Yaskawa INFORM job: big_bent_cylinder_program.JBI

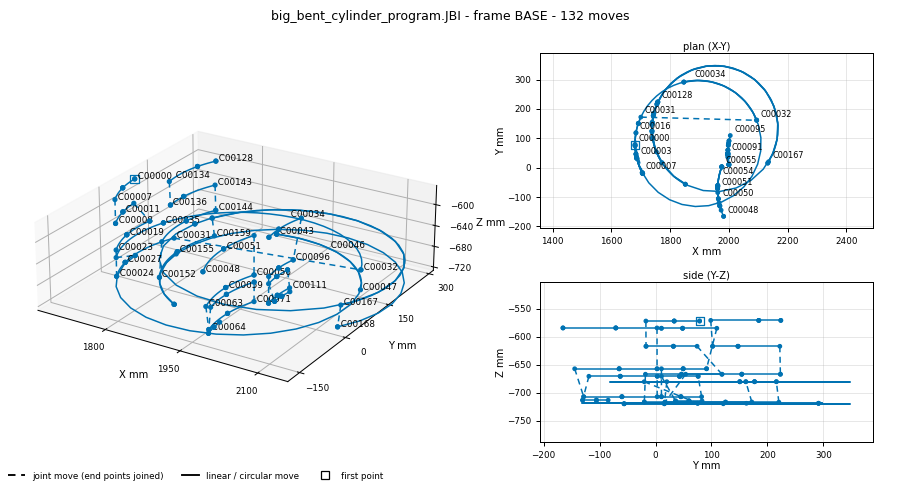
[picture p0: tool path of big_bent_cylinder_program.JBI in frame BASE, 132 of 185 moves have a stored position in this frame; points joined in program order, loops and branches not executed]
/JOB
//NAME big_bent_cylinder_program
//POS
///NPOS 176,0,176,0,0,0
///TOOL 0
///POSTYPE BASE
///RECTAN
///RCONF 0,0,0,0,0,0,0,0,0,0,0,0,0,0,0,0,0,0,0,0,0,0,0,0
C00000=1680.662060,78.729011,-571.725500,-175.000000,-89.999999,5.000000
C00001=1680.662060,78.729011,-571.725500,-175.000000,-89.999999,5.000000
C00002=1681.281377,65.697405,-571.725500,-175.000000,-89.999999,5.000000
C00003=1686.307736,33.361169,-571.725500,-166.791969,-90.000000,5.000000
C00004=1686.307736,33.361169,-571.725500,-166.791969,-90.000000,5.000000
C00005=1686.307736,33.361169,-571.725500,-166.791969,-90.000000,5.000000
C00006=1696.081532,2.440055,-571.725500,-158.125782,-90.000000,5.000000
C00007=1705.179944,-17.274311,-571.725500,-152.326458,-90.000000,5.000000
C00008=1705.056434,-17.038439,-616.865500,-152.397542,-90.000000,5.000000
C00009=1705.056434,-17.038439,-616.865500,-152.397542,-90.000000,5.000000
C00010=1691.809992,14.034424,-616.865500,-161.425103,-90.000000,5.000000
C00011=1686.649002,31.929188,-616.865500,-166.398950,-89.999999,5.000000
C00012=1686.649002,31.929188,-616.865500,-166.398950,-89.999999,5.000000
C00013=1686.649002,31.929188,-616.865500,-166.398950,-89.999999,5.000000
C00014=1685.912600,35.076369,-616.865500,-167.261890,-89.999999,5.000000
C00015=1680.785043,74.259067,-616.865500,-175.000000,-89.999999,5.000000
C00016=1683.724650,118.705496,-666.897500,170.259212,-90.000000,5.000000
C00017=1683.724650,118.705496,-666.897500,170.259212,-90.000000,5.000000
C00018=1682.076679,57.525758,-666.897500,-173.345168,-90.000000,5.000000
C00019=1683.676867,46.365991,-666.897500,-170.334905,-89.999999,5.000000
C00020=1683.676867,46.365991,-666.897500,-170.334905,-89.999999,5.000000
C00021=1683.676867,46.365991,-666.897500,-170.334905,-89.999999,5.000000
C00022=1694.919230,5.398308,-666.897500,-158.974360,-90.000000,5.000000
C00023=1705.611428,-18.092796,-666.897500,-152.079433,-90.000000,5.000000
C00024=1706.664513,-20.055320,-716.487000,-151.484806,-89.999999,5.000000
C00025=1706.664513,-20.055320,-716.487000,-151.484806,-89.999999,5.000000
C00026=1685.911416,35.081606,-716.487000,-167.263323,-89.999999,5.000000
C00027=1685.559141,36.668028,-716.487000,-167.697185,-90.000000,5.000000
C00028=1685.559141,36.668028,-716.487000,-167.697185,-90.000000,5.000000
C00029=1685.559141,36.668028,-716.487000,-167.697185,-90.000000,5.000000
C00030=1681.109891,96.728954,-716.487000,175.000000,-90.000000,5.000000
C00031=1700.273814,172.091124,-716.487000,155.294663,-89.999999,5.000000
C00032=2094.761755,161.426578,-680.269460,175.000000,-60.000000,-158.391764
C00033=2094.761755,161.426578,-680.269460,175.000000,-60.000000,-158.391764
C00034=1868.772286,295.364365,-680.269460,-175.000000,-60.000000,-82.916364
C00035=1691.784994,150.683171,-680.269460,175.000000,-60.000000,-18.553935
C00036=1691.784994,150.683171,-680.269460,175.000000,-60.000000,-18.553935
C00037=1691.784994,150.683171,-680.269460,175.000000,-60.000000,-18.553935
C00038=1682.232356,108.566108,-680.269460,175.000000,-60.000000,-7.004345
C00039=1706.777106,-20.262288,-680.269460,175.000000,-60.000000,28.578098
C00040=1680.746964,75.333699,-718.844460,175.000000,-60.000000,5.000000
C00041=1680.746964,75.333699,-718.844460,175.000000,-60.000000,5.000000
C00042=1686.705940,31.694430,-718.844460,175.000000,-60.000000,13.665543
C00043=1846.719133,291.446034,-718.844460,-175.000000,-60.000000,-76.933666
C00044=1846.719133,291.446034,-718.844460,-175.000000,-60.000000,-76.933666
C00045=1846.719133,291.446034,-718.844460,-175.000000,-60.000000,-76.933666
C00046=1958.496559,287.467102,-718.844460,-175.000000,-60.000000,-107.143719
C00047=2094.352293,162.452606,-718.844460,175.000000,-60.000000,-158.096827
C00048=1982.067357,-165.559936,-584.093000,-155.080908,-90.000000,5.000000
C00049=1982.067357,-165.559936,-584.093000,-155.080908,-90.000000,5.000000
C00050=1964.611411,-108.659635,-584.093000,-170.809028,-89.999999,5.000000
C00051=1961.837117,-71.115701,-584.093000,175.000000,-90.000000,5.000000
C00052=1961.837117,-71.115701,-584.093000,175.000000,-90.000000,5.000000
C00053=1961.837117,-71.115701,-584.093000,175.000000,-90.000000,5.000000
C00054=1965.708987,-32.968576,-584.093000,169.147482,-90.000000,5.000000
C00055=1975.726992,2.608125,-584.093000,159.399257,-90.000000,5.000000
C00056=1975.761045,2.698658,-657.086000,159.373776,-90.000000,5.000000
C00057=1975.761045,2.698658,-657.086000,159.373776,-90.000000,5.000000
C00058=1965.914945,-31.908497,-657.086000,168.863002,-90.000000,5.000000
C00059=1961.998779,-65.079199,-657.086000,175.000000,-90.000000,5.000000
C00060=1961.998779,-65.079199,-657.086000,175.000000,-90.000000,5.000000
C00061=1961.998779,-65.079199,-657.086000,175.000000,-90.000000,5.000000
C00062=1963.509319,-100.982572,-657.086000,-172.852243,-90.000000,5.000000
C00063=1973.616747,-144.579151,-657.086000,-161.042059,-90.000000,5.000000
C00064=1968.783955,-128.519960,-707.081000,-165.461049,-90.000000,5.000000
C00065=1968.783955,-128.519960,-707.081000,-165.461049,-90.000000,5.000000
C00066=1962.624689,-92.622591,-707.081000,-175.000000,-89.999999,5.000000
C00067=1962.256000,-60.139714,-707.081000,175.000000,-89.999999,5.000000
C00068=1962.256000,-60.139714,-707.081000,175.000000,-89.999999,5.000000
C00069=1962.256000,-60.139714,-707.081000,175.000000,-89.999999,5.000000
C00070=1966.568329,-28.715907,-707.081000,168.004536,-90.000000,5.000000
C00071=1975.822267,2.861113,-707.081000,159.328043,-90.000000,5.000000
C00072=1975.889379,3.038750,-670.514960,175.000000,-60.000000,-20.721981
C00073=1975.889379,3.038750,-670.514960,175.000000,-60.000000,-20.721981
C00074=1966.483865,-29.115276,-670.514960,-175.000000,-60.000000,-11.887931
C00075=1962.086887,-63.128851,-670.514960,-175.000000,-60.000000,-5.000000
C00076=1962.086887,-63.128851,-670.514960,-175.000000,-60.000000,-5.000000
C00077=1962.086887,-63.128851,-670.514960,-175.000000,-60.000000,-5.000000
C00078=1962.474161,-90.788003,-670.514960,175.000000,-60.000000,5.000000
C00079=1966.582713,-119.190828,-670.514960,175.000000,-60.000000,12.013682
C00080=1969.287032,-130.424250,-713.241460,-175.000000,-60.000000,15.057812
C00081=1969.287032,-130.424250,-713.241460,-175.000000,-60.000000,15.057812
C00082=1965.276012,-112.543631,-713.241460,175.000000,-60.000000,10.229021
C00083=1964.157808,-105.729691,-713.241460,175.000000,-60.000000,8.409934
C00084=1964.157808,-105.729691,-713.241460,175.000000,-60.000000,8.409934
C00085=1964.157808,-105.729691,-713.241460,175.000000,-60.000000,8.409934
C00086=1963.054065,-97.064846,-713.241460,175.000000,-60.000000,6.108749
C00087=1962.089517,-84.763052,-713.241460,175.000000,-60.000000,5.000000
C00088=2000.069543,10.498430,-584.670000,-169.548727,-90.000000,5.000000
C00089=2000.069543,10.498430,-584.670000,-169.548727,-90.000000,5.000000
C00090=1997.571310,28.005118,-584.670000,-174.208531,-90.000000,5.000000
C00091=1996.467025,48.352787,-584.670000,-175.000000,-90.000000,5.000000
C00092=1996.467025,48.352787,-584.670000,-175.000000,-90.000000,5.000000
C00093=1996.467025,48.352787,-584.670000,-175.000000,-90.000000,5.000000
C00094=1997.381403,69.939092,-584.670000,174.727478,-90.000000,5.000000
C00095=2004.784425,109.545499,-584.670000,164.098004,-90.000000,5.000000
C00096=2000.404432,91.180757,-657.053500,169.073094,-89.999999,5.000000
C00097=2000.404432,91.180757,-657.053500,169.073094,-89.999999,5.000000
C00098=1997.278351,68.789047,-657.053500,175.000000,-90.000000,5.000000
C00099=1996.461833,49.404029,-657.053500,-175.000000,-89.999999,5.000000
C00100=1996.461833,49.404029,-657.053500,-175.000000,-89.999999,5.000000
C00101=1996.461833,49.404029,-657.053500,-175.000000,-89.999999,5.000000
C00102=1997.397112,29.796400,-657.053500,-174.682637,-89.999999,5.000000
C00103=2000.060639,10.546731,-657.053500,-169.561666,-90.000000,5.000000
C00104=2000.066177,10.516684,-707.079500,-169.553617,-90.000000,5.000000
C00105=2000.066177,10.516684,-707.079500,-169.553617,-90.000000,5.000000
C00106=1997.595455,27.768350,-707.079500,-174.145835,-90.000000,5.000000
C00107=1996.509510,45.365815,-707.079500,-175.000000,-90.000000,5.000000
C00108=1996.509510,45.365815,-707.079500,-175.000000,-90.000000,5.000000
C00109=1996.509510,45.365815,-707.079500,-175.000000,-90.000000,5.000000
C00110=1996.804625,62.171171,-707.079500,175.000000,-89.999999,5.000000
C00111=1998.889041,82.359813,-707.079500,171.431009,-90.000000,5.000000
C00112=1998.045406,76.156312,-670.596960,175.000000,-60.000000,-6.919699
C00113=1998.045406,76.156312,-670.596960,175.000000,-60.000000,-6.919699
C00114=1996.569713,56.823909,-670.596960,175.000000,-60.000000,-5.000000
C00115=1996.576887,42.857740,-670.596960,-175.000000,-60.000000,5.000000
C00116=1996.576887,42.857740,-670.596960,-175.000000,-60.000000,5.000000
C00117=1996.576887,42.857740,-670.596960,-175.000000,-60.000000,5.000000
C00118=1997.640727,27.331167,-670.596960,175.000000,-60.000000,5.969948
C00119=2000.064475,10.525917,-670.596960,-175.000000,-60.000000,10.443910
C00120=1996.926560,35.731421,-714.596460,-175.000000,-60.000000,5.000000
C00121=1996.926560,35.731421,-714.596460,-175.000000,-60.000000,5.000000
C00122=1996.461166,50.054368,-714.596460,-175.000000,-60.000000,-5.000000
C00123=1996.686893,59.859568,-714.596460,175.000000,-60.000000,-5.000000
C00124=1996.686893,59.859568,-714.596460,175.000000,-60.000000,-5.000000
C00125=1996.686893,59.859568,-714.596460,175.000000,-60.000000,-5.000000
C00126=1997.059270,66.071625,-714.596460,175.000000,-60.000000,-5.000000
C00127=1998.999277,83.083128,-714.596460,-175.000000,-60.000000,-8.761734
C00128=1758.269028,223.964920,-570.597000,154.967152,-89.999999,5.000000
C00129=1758.269028,223.964920,-570.597000,154.967152,-89.999999,5.000000
C00130=1747.306451,195.306976,-570.597000,163.165957,-90.000000,5.000000
C00131=1744.365779,184.595198,-570.597000,166.131935,-90.000000,5.000000
C00132=1744.365779,184.595198,-570.597000,166.131935,-90.000000,5.000000
C00133=1744.365779,184.595198,-570.597000,166.131935,-90.000000,5.000000
C00134=1738.882687,114.962659,-570.597000,-175.000000,-90.000000,5.000000
C00135=1740.902973,98.646591,-570.597000,-170.746248,-90.000000,5.000000
C00136=1740.380838,102.020143,-616.899000,-171.657655,-89.999999,5.000000
C00137=1740.380838,102.020143,-616.899000,-171.657655,-89.999999,5.000000
C00138=1740.368462,102.104660,-616.899000,-171.680460,-90.000000,5.000000
C00139=1738.585922,147.440519,-616.899000,175.000000,-90.000000,5.000000
C00140=1738.585922,147.440519,-616.899000,175.000000,-90.000000,5.000000
C00141=1738.585922,147.440519,-616.899000,175.000000,-90.000000,5.000000
C00142=1740.437140,164.675109,-616.899000,171.554682,-90.000000,5.000000
C00143=1757.452118,222.194741,-616.899000,155.487655,-89.999999,5.000000
C00144=1757.925437,223.225529,-666.848500,155.184828,-90.000000,5.000000
C00145=1757.925437,223.225529,-666.848500,155.184828,-90.000000,5.000000
C00146=1746.009027,190.845212,-666.848500,164.406527,-89.999999,5.000000
C00147=1739.139294,154.149814,-666.848500,174.386304,-89.999999,5.000000
C00148=1739.139294,154.149814,-666.848500,174.386304,-89.999999,5.000000
C00149=1739.139294,154.149814,-666.848500,174.386304,-89.999999,5.000000
C00150=1738.284639,124.502088,-666.848500,-175.000000,-89.999999,5.000000
C00151=1753.300912,53.851424,-666.848500,-158.312815,-90.000000,5.000000
C00152=1772.394009,16.796526,-716.805500,-147.166240,-90.000000,5.000000
C00153=1772.394009,16.796526,-716.805500,-147.166240,-90.000000,5.000000
C00154=1739.108172,112.482950,-716.805500,-174.471895,-90.000000,5.000000
C00155=1738.260942,125.110643,-716.805500,-175.000000,-90.000000,5.000000
C00156=1738.260942,125.110643,-716.805500,-175.000000,-90.000000,5.000000
C00157=1738.260942,125.110643,-716.805500,-175.000000,-90.000000,5.000000
C00158=1742.358990,175.649731,-716.805500,168.579748,-90.000000,5.000000
C00159=1756.674616,220.469533,-716.805500,155.992868,-89.999999,5.000000
C00160=1754.756309,216.028366,-680.232460,175.000000,-60.000000,-22.715517
C00161=1754.756309,216.028366,-680.232460,175.000000,-60.000000,-22.715517
C00162=1738.200104,139.373252,-680.232460,175.000000,-60.000000,-5.000000
C00163=1742.647823,177.055343,-680.232460,175.000000,-60.000000,-11.803365
C00164=1742.647823,177.055343,-680.232460,175.000000,-60.000000,-11.803365
C00165=1742.647823,177.055343,-680.232460,175.000000,-60.000000,-11.803365
C00166=1751.432629,207.592922,-680.232460,175.000000,-60.000000,-20.294724
C00167=2135.172444,20.171370,-680.232460,175.000000,-60.000000,148.232228
C00168=2132.324586,15.696959,-719.653460,175.000000,-60.000000,146.816171
C00169=2132.324586,15.696959,-719.653460,175.000000,-60.000000,146.816171
C00170=1752.153842,209.514861,-719.653460,175.000000,-60.000000,-20.842785
C00171=1851.714259,-56.195906,-719.653460,-175.000000,-60.000000,61.924201
C00172=1851.714259,-56.195906,-719.653460,-175.000000,-60.000000,61.924201
C00173=1851.714259,-56.195906,-719.653460,-175.000000,-60.000000,61.924201
C00174=1751.649749,58.136260,-719.653460,175.000000,-60.000000,20.461195
C00175=1738.447744,121.122397,-719.653460,175.000000,-60.000000,5.000000
///POSTYPE PULSE
///PULSE
EX00000=26624.0
EX00001=162816.0
EX00002=194560.0
EX00003=340992.0
///POSTYPE PULSE
///PULSE
EC00000=26624.0
EC00001=26624.0
EC00002=26624.0
EC00003=26624.0
EC00004=26624.0
EC00005=26624.0
EC00006=26624.0
EC00007=26624.0
EC00008=26624.0
EC00009=26624.0
EC00010=26624.0
EC00011=26624.0
EC00012=26624.0
EC00013=26624.0
EC00014=26624.0
EC00015=26624.0
EC00016=26624.0
EC00017=26624.0
EC00018=26624.0
EC00019=26624.0
EC00020=26624.0
EC00021=26624.0
EC00022=26624.0
EC00023=26624.0
EC00024=26624.0
EC00025=26624.0
EC00026=26624.0
EC00027=26624.0
EC00028=26624.0
EC00029=26624.0
EC00030=26624.0
EC00031=26624.0
EC00032=26624.0
EC00033=26624.0
EC00034=26624.0
EC00035=26624.0
EC00036=26624.0
EC00037=26624.0
EC00038=26624.0
EC00039=26624.0
EC00040=26624.0
EC00041=26624.0
EC00042=26624.0
EC00043=26624.0
EC00044=26624.0
EC00045=26624.0
EC00046=26624.0
EC00047=26624.0
EC00048=162816.0
EC00049=162816.0
EC00050=162816.0
EC00051=162816.0
EC00052=162816.0
EC00053=162816.0
EC00054=162816.0
EC00055=162816.0
EC00056=162816.0
EC00057=162816.0
EC00058=162816.0
EC00059=162816.0
EC00060=162816.0
EC00061=162816.0
EC00062=162816.0
EC00063=162816.0
EC00064=162816.0
EC00065=162816.0
EC00066=162816.0
EC00067=162816.0
EC00068=162816.0
EC00069=162816.0
EC00070=162816.0
EC00071=162816.0
EC00072=162816.0
EC00073=162816.0
EC00074=162816.0
EC00075=162816.0
EC00076=162816.0
EC00077=162816.0
EC00078=162816.0
EC00079=162816.0
EC00080=162816.0
EC00081=162816.0
EC00082=162816.0
EC00083=162816.0
EC00084=162816.0
EC00085=162816.0
EC00086=162816.0
EC00087=162816.0
EC00088=194560.0
EC00089=194560.0
EC00090=194560.0
EC00091=194560.0
EC00092=194560.0
EC00093=194560.0
EC00094=194560.0
EC00095=194560.0
EC00096=194560.0
EC00097=194560.0
EC00098=194560.0
EC00099=194560.0
EC00100=194560.0
EC00101=194560.0
EC00102=194560.0
EC00103=194560.0
EC00104=194560.0
EC00105=194560.0
EC00106=194560.0
EC00107=194560.0
EC00108=194560.0
EC00109=194560.0
EC00110=194560.0
EC00111=194560.0
EC00112=194560.0
EC00113=194560.0
EC00114=194560.0
EC00115=194560.0
EC00116=194560.0
EC00117=194560.0
EC00118=194560.0
EC00119=194560.0
EC00120=194560.0
EC00121=194560.0
EC00122=194560.0
EC00123=194560.0
EC00124=194560.0
EC00125=194560.0
EC00126=194560.0
EC00127=194560.0
EC00128=340992.0
EC00129=340992.0
EC00130=340992.0
EC00131=340992.0
EC00132=340992.0
EC00133=340992.0
EC00134=340992.0
EC00135=340992.0
EC00136=340992.0
EC00137=340992.0
EC00138=340992.0
EC00139=340992.0
EC00140=340992.0
EC00141=340992.0
EC00142=340992.0
EC00143=340992.0
EC00144=340992.0
EC00145=340992.0
EC00146=340992.0
EC00147=340992.0
EC00148=340992.0
EC00149=340992.0
EC00150=340992.0
EC00151=340992.0
EC00152=340992.0
EC00153=340992.0
EC00154=340992.0
EC00155=340992.0
EC00156=340992.0
EC00157=340992.0
EC00158=340992.0
EC00159=340992.0
EC00160=340992.0
EC00161=340992.0
EC00162=340992.0
EC00163=340992.0
EC00164=340992.0
EC00165=340992.0
EC00166=340992.0
EC00167=340992.0
EC00168=340992.0
EC00169=340992.0
EC00170=340992.0
EC00171=340992.0
EC00172=340992.0
EC00173=340992.0
EC00174=340992.0
EC00175=340992.0
//INST
///DATE 2023/08/16 12:18
///ATTR SC,RW,RJ
////FRAME BASE
///GROUP1 RB1,ST1
NOP
MOVJ P009 EX000 VJ=15.00
MOVJ C00000 EC00000 VJ=15.0
CALL JOB:SPYON
MOVC C00001 EC00001 V=150.0
MOVC C00002 EC00002 V=150.0
MOVC C00003 EC00003 V=150.0
MOVJ C00004 EC00004 VJ=15.0
MOVC C00005 EC00005 V=150.0
MOVC C00006 EC00006 V=150.0
MOVC C00007 EC00007 V=150.0
MOVJ C00008 EC00008 VJ=15.0
MOVC C00009 EC00009 V=150.0
MOVC C00010 EC00010 V=150.0
MOVC C00011 EC00011 V=150.0
MOVJ C00012 EC00012 VJ=15.0
MOVC C00013 EC00013 V=150.0
MOVC C00014 EC00014 V=150.0
MOVC C00015 EC00015 V=150.0
MOVJ C00016 EC00016 VJ=15.0
MOVC C00017 EC00017 V=150.0
MOVC C00018 EC00018 V=150.0
MOVC C00019 EC00019 V=150.0
MOVJ C00020 EC00020 VJ=15.0
MOVC C00021 EC00021 V=150.0
MOVC C00022 EC00022 V=150.0
MOVC C00023 EC00023 V=150.0
MOVJ C00024 EC00024 VJ=15.0
MOVC C00025 EC00025 V=150.0
MOVC C00026 EC00026 V=150.0
MOVC C00027 EC00027 V=150.0
MOVJ C00028 EC00028 VJ=15.0
MOVC C00029 EC00029 V=150.0
MOVC C00030 EC00030 V=150.0
MOVC C00031 EC00031 V=150.0
MOVJ C00032 EC00032 VJ=15.0
MOVC C00033 EC00033 V=150.0
MOVC C00034 EC00034 V=150.0
MOVC C00035 EC00035 V=150.0
MOVJ C00036 EC00036 VJ=15.0
MOVC C00037 EC00037 V=150.0
MOVC C00038 EC00038 V=150.0
MOVC C00039 EC00039 V=150.0
MOVJ C00040 EC00040 VJ=15.0
MOVC C00041 EC00041 V=150.0
MOVC C00042 EC00042 V=150.0
MOVC C00043 EC00043 V=150.0
MOVJ C00044 EC00044 VJ=15.0
MOVC C00045 EC00045 V=150.0
MOVC C00046 EC00046 V=150.0
MOVC C00047 EC00047 V=150.0
CALL JOB:SPYOF
MOVJ P009 VJ=15.00
MOVL P009 EX00000 V=150.0
MOVJ C00048 EC00048 VJ=15.0
CALL JOB:SPYON
MOVC C00049 EC00049 V=150.0
MOVC C00050 EC00050 V=150.0
MOVC C00051 EC00051 V=150.0
MOVJ C00052 EC00052 VJ=15.0
MOVC C00053 EC00053 V=150.0
MOVC C00054 EC00054 V=150.0
MOVC C00055 EC00055 V=150.0
MOVJ C00056 EC00056 VJ=15.0
MOVC C00057 EC00057 V=150.0
MOVC C00058 EC00058 V=150.0
MOVC C00059 EC00059 V=150.0
MOVJ C00060 EC00060 VJ=15.0
MOVC C00061 EC00061 V=150.0
MOVC C00062 EC00062 V=150.0
MOVC C00063 EC00063 V=150.0
MOVJ C00064 EC00064 VJ=15.0
MOVC C00065 EC00065 V=150.0
MOVC C00066 EC00066 V=150.0
MOVC C00067 EC00067 V=150.0
MOVJ C00068 EC00068 VJ=15.0
MOVC C00069 EC00069 V=150.0
MOVC C00070 EC00070 V=150.0
MOVC C00071 EC00071 V=150.0
MOVJ C00072 EC00072 VJ=15.0
MOVC C00073 EC00073 V=150.0
MOVC C00074 EC00074 V=150.0
MOVC C00075 EC00075 V=150.0
MOVJ C00076 EC00076 VJ=15.0
MOVC C00077 EC00077 V=150.0
MOVC C00078 EC00078 V=150.0
MOVC C00079 EC00079 V=150.0
MOVJ C00080 EC00080 VJ=15.0
MOVC C00081 EC00081 V=150.0
MOVC C00082 EC00082 V=150.0
MOVC C00083 EC00083 V=150.0
MOVJ C00084 EC00084 VJ=15.0
MOVC C00085 EC00085 V=150.0
MOVC C00086 EC00086 V=150.0
MOVC C00087 EC00087 V=150.0
CALL JOB:SPYOF
MOVJ P009 VJ=15.00
MOVL P009 EX00001 V=150.0
MOVJ C00088 EC00088 VJ=15.0
CALL JOB:SPYON
MOVC C00089 EC00089 V=150.0
MOVC C00090 EC00090 V=150.0
MOVC C00091 EC00091 V=150.0
MOVJ C00092 EC00092 VJ=15.0
MOVC C00093 EC00093 V=150.0
MOVC C00094 EC00094 V=150.0
MOVC C00095 EC00095 V=150.0
MOVJ C00096 EC00096 VJ=15.0
MOVC C00097 EC00097 V=150.0
MOVC C00098 EC00098 V=150.0
MOVC C00099 EC00099 V=150.0
MOVJ C00100 EC00100 VJ=15.0
MOVC C00101 EC00101 V=150.0
MOVC C00102 EC00102 V=150.0
MOVC C00103 EC00103 V=150.0
MOVJ C00104 EC00104 VJ=15.0
MOVC C00105 EC00105 V=150.0
MOVC C00106 EC00106 V=150.0
MOVC C00107 EC00107 V=150.0
MOVJ C00108 EC00108 VJ=15.0
MOVC C00109 EC00109 V=150.0
MOVC C00110 EC00110 V=150.0
MOVC C00111 EC00111 V=150.0
MOVJ C00112 EC00112 VJ=15.0
MOVC C00113 EC00113 V=150.0
MOVC C00114 EC00114 V=150.0
MOVC C00115 EC00115 V=150.0
MOVJ C00116 EC00116 VJ=15.0
MOVC C00117 EC00117 V=150.0
MOVC C00118 EC00118 V=150.0
MOVC C00119 EC00119 V=150.0
MOVJ C00120 EC00120 VJ=15.0
MOVC C00121 EC00121 V=150.0
MOVC C00122 EC00122 V=150.0
MOVC C00123 EC00123 V=150.0
MOVJ C00124 EC00124 VJ=15.0
MOVC C00125 EC00125 V=150.0
MOVC C00126 EC00126 V=150.0
MOVC C00127 EC00127 V=150.0
CALL JOB:SPYOF
MOVJ P009 VJ=15.00
MOVL P009 EX00002 V=150.0
MOVJ C00128 EC00128 VJ=15.0
CALL JOB:SPYON
MOVC C00129 EC00129 V=150.0
MOVC C00130 EC00130 V=150.0
MOVC C00131 EC00131 V=150.0
MOVJ C00132 EC00132 VJ=15.0
MOVC C00133 EC00133 V=150.0
MOVC C00134 EC00134 V=150.0
MOVC C00135 EC00135 V=150.0
MOVJ C00136 EC00136 VJ=15.0
MOVC C00137 EC00137 V=150.0
MOVC C00138 EC00138 V=150.0
MOVC C00139 EC00139 V=150.0
MOVJ C00140 EC00140 VJ=15.0
MOVC C00141 EC00141 V=150.0
MOVC C00142 EC00142 V=150.0
MOVC C00143 EC00143 V=150.0
MOVJ C00144 EC00144 VJ=15.0
MOVC C00145 EC00145 V=150.0
MOVC C00146 EC00146 V=150.0
MOVC C00147 EC00147 V=150.0
MOVJ C00148 EC00148 VJ=15.0
MOVC C00149 EC00149 V=150.0
MOVC C00150 EC00150 V=150.0
MOVC C00151 EC00151 V=150.0
MOVJ C00152 EC00152 VJ=15.0
MOVC C00153 EC00153 V=150.0
MOVC C00154 EC00154 V=150.0
MOVC C00155 EC00155 V=150.0
MOVJ C00156 EC00156 VJ=15.0
MOVC C00157 EC00157 V=150.0
MOVC C00158 EC00158 V=150.0
MOVC C00159 EC00159 V=150.0
MOVJ C00160 EC00160 VJ=15.0
MOVC C00161 EC00161 V=150.0
MOVC C00162 EC00162 V=150.0
MOVC C00163 EC00163 V=150.0
MOVJ C00164 EC00164 VJ=15.0
MOVC C00165 EC00165 V=150.0
MOVC C00166 EC00166 V=150.0
MOVC C00167 EC00167 V=150.0
MOVJ C00168 EC00168 VJ=15.0
MOVC C00169 EC00169 V=150.0
MOVC C00170 EC00170 V=150.0
MOVC C00171 EC00171 V=150.0
MOVJ C00172 EC00172 VJ=15.0
MOVC C00173 EC00173 V=150.0
MOVC C00174 EC00174 V=150.0
MOVC C00175 EC00175 V=150.0
CALL JOB:SPYOF
MOVJ P009 VJ=15.00
MOVL P009 EX00003 V=150.0
END
